TYPE WordToBytes :
UNION
	word_in			: WORD;
	bytes			: ARRAY [0..1] OF BYTE;
END_UNION
END_TYPE

(* stored: Version 1.1.0.1, ProductVersion 3.1.4024.11
   DUT WordToBytes: Id {4d03d9da-9ed3-4725-b621-03f2fc74b961} *)
